//Encoder reference positions for MR4K2
nEncRefXM4K2  := ULINT_TO_UDINT(GVL_M4K2.nM4K2X_ENC_REF);
nEncRefYM4K2  := ULINT_TO_UDINT(GVL_M4K2.nM4K2Y_ENC_REF);
nEncRefrXM4K2  := ULINT_TO_UDINT(GVL_M4K2.nM4K2rX_ENC_REF);
nEncRefUSM4K2  := ULINT_TO_UDINT(GVL_M4K2.nM4K2US_ENC_REF);
nEncRefDSM4K2  := ULINT_TO_UDINT(GVL_M4K2.nM4K2DS_ENC_REF);

// M4K2 Bender Encoder Count Values For Epics
nEncCntXM4K2  := ULINT_TO_UDINT(M33.nRawEncoderULINT);
nEncCntYM4K2  := ULINT_TO_UDINT(M34.nRawEncoderULINT);
nEncCntrXM4K2  := ULINT_TO_UDINT(M35.nRawEncoderULINT);
nEncCntUSM4K2  := ULINT_TO_UDINT(M36.nRawEncoderULINT);
nEncCntDSM4K2  := ULINT_TO_UDINT(M37.nRawEncoderULINT);

// MR4K2 Bender RTDs
fM4K2US_RTD_1 := INT_TO_REAL(GVL_M4K2.nM4K2US_RTD_1);
fM4K2US_RTD_2 := INT_TO_REAL(GVL_M4K2.nM4K2US_RTD_2);
fM4K2US_RTD_3 := INT_TO_REAL(GVL_M4K2.nM4K2US_RTD_3);

fM4K2DS_RTD_1 := INT_TO_REAL(GVL_M4K2.nM4K2DS_RTD_1);


// RTD not connected if T=0
bM4K2US_RTD_1_Err := fM4K2US_RTD_1 = 0;
bM4K2US_RTD_2_Err := fM4K2US_RTD_2 = 0;
bM4K2US_RTD_3_Err := fM4K2US_RTD_3 = 0;
bM4K2DS_RTD_1_Err := fM4K2DS_RTD_1 = 0;

// M4K2 Bender RTD interlocks
M36.bHardwareEnable R= fM4K2US_RTD_1 > 9000 OR bM4K2US_RTD_1_Err;
M37.bHardwareEnable R= fM4K2DS_RTD_1 > 9000 OR bM4K2DS_RTD_1_Err;

fbM4K2_Chin_Right_RTD(fResolution:=0.01);
fbM4K2_Chin_Left_RTD(fResolution:=0.01);

// Axilon Cooling Panel
fbCoolingPanel();
(*
//PMPS
ffBenderRange.i_xOK :=
    GVL_M4K2.nM4K2US_PMPS_LowerLimit < nEncCntUSM4K2 AND nEncCntUSM4K2 < GVL_M4K2.nM4K2US_PMPS_UpperLimit AND
    GVL_M4K2.nM4K2DS_PMPS_LowerLimit < nEncCntDSM4K2 AND nEncCntUSM4K2 < GVL_M4K2.nM4K2DS_PMPS_UpperLimit;
ffBenderRange(io_fbFFHWO := GVL_PMPS.fbFastFaultOutput1);
*)
fbXSetup(stPositionState:=GVL_States.stDefaultKBX, bSetDefault:=TRUE);

fbXSetup(stPositionState:=astCoatingStatesX[E_B4C_Rh_CoatingStates.B4C],
    sName:='B4C',
    sPmpsState:='MR4K2:KBV-B4C',
    nEncoderCount:=5824240,
    fDelta:=5
);
fbXSetup(stPositionState:=astCoatingStatesX[E_B4C_Rh_CoatingStates.Rh],
    sName:='Rh',
    sPmpsState:='MR4K2:KBV-RHODIUM',
    nEncoderCount:=3524222,
    fDelta:=1.5
);
fbCoatingStates(
    stMotionStage:=Main.M33,
    astPositionState:=astCoatingStatesX,
    eEnumSet:=eStateSet,
    eEnumGet:=eStateGet,
    fbFFHWO:=GVL_PMPS.fbFastFaultOutput2,
    fbArbiter:=GVL_PMPS.fbArbiter2,
    bEnableMotion:=TRUE,
    bEnableBeamParams:=TRUE,
    sDeviceName:='MR4K2:KBV',
    sTransitionKey:='MR4K2:KBV-TRANSITION',
);

END_PROGRAM

// ---- POUs/Serial Comm/P_Serial_Com.TcPOU
PROGRAM P_Serial_Com
VAR
    fbSerialLineControl_EL6001_M1K2: SerialLineControl;
END_VAR

//These are the global IOs...don't forget to copy your data into them

(* EL6001 Serial port 0 com function *)
fbSerialLineControl_EL6001_M1K2(Mode:= SERIALLINEMODE_EL6_22B (*SERIALLINEMODE_KL6_22B_STANDARD*),
                                pComIn:= ADR(Serial_stComIn_M1K2),
                                   pComOut:=ADR(Serial_stComOut_M1K2),
                                SizeComIn:= SIZEOF(Serial_stComIn_M1K2),
                                TxBuffer:= Serial_TXBuffer_M1K2,
                                RxBuffer:= Serial_RXBuffer_M1K2,
                                Error=> ,
                                ErrorID=> );

END_PROGRAM

// ---- POUs/PRG_Stats.TcPOU
PROGRAM PRG_Stats
VAR
    // SP1K1 Grating Mono Vibration Stats
    fGpiEncoderPosDiff: LREAL;
    afGpiPosDiffBuffer: ARRAY[1..1000] OF LREAL;
    afGpiExtraBuffer: ARRAY[1..1000] OF LREAL;
    fbGpiPosDiffCollect: FB_DataBuffer;
    {attribute 'pytmc' := '
        pv: SP1K1:MONO:MMS:G_PI:ENCDIFF
    '}
    fbGpiPosDiffStats: FB_BasicStats;

    fGpiRangeMax: LREAL;
    rtNewGpiMove: R_TRIG;
    tonNewGpiMove: TON;


    // SP1K1 Mirror Pitch Mono Vibration Stats
    fMpiEncoderPosDiff: LREAL;
    afMpiPosDiffBuffer: ARRAY[1..1000] OF LREAL;
    afMpiExtraBuffer: ARRAY[1..1000] OF LREAL;
    fbMpiPosDiffCollect: FB_DataBuffer;
    {attribute 'pytmc' := '
        pv: SP1K1:MONO:MMS:M_PI:ENCDIFF
    '}
    fbMpiPosDiffStats: FB_BasicStats;


    // MR1K1 Pitch Vibration Stats
    fMR1K1PiEncoderPosDiff: LREAL;
    afMR1K1PiPosDiffBuffer: ARRAY[1..1000] OF LREAL;
    afMR1K1PiExtraBuffer: ARRAY[1..1000] OF LREAL;
    fbMR1K1PiPosDiffCollect: FB_DataBuffer;
    {attribute 'pytmc' := '
        pv: MR1K1:BEND:MMS:PITCH:ENCDIFF
    '}
    fbMR1K1PiPosDiffStats: FB_BasicStats;
END_VAR

IF rtNewGpiMove.Q THEN
    // Reset before a move
    fGpiRangeMax := 0;
ELSIF tonNewGpiMove.Q AND ABS(M7.fPosition - M7.stAxisStatus.fActPosition) > 5 THEN
    // Update only during moves, not at the start or end
    fGpiRangeMax := MAX(fGpiRangeMax, fbGpiPosDiffStats.fRange);
END_IF

fGpiEncoderPosDiff := ((UDINT_TO_LREAL(M7.nEncoderCount) / 150.0) - (M7.Axis.NcToPlc.SetPos - M7.stAxisParameters.fEncOffset)) * 1000;
fbGpiPosDiffCollect(
    bExecute:=TRUE,
    pInputAdr:=ADR(fGpiEncoderPosDiff),
    iInputSize:=SIZEOF(fGpiEncoderPosDiff),
    iElemCount:=1000,
    pPartialAdr:=ADR(afGpiPosDiffBuffer),
    pOutputAdr:=ADR(afGpiExtraBuffer),
);
fbGpiPosDiffStats(
    aSignal:=afGpiPosDiffBuffer,
    bAlwaysCalc:=TRUE,
);
rtNewGpiMove(CLK:=M7.bExecute);
tonNewGpiMove(
    IN:=M7.bExecute,
    PT:=T#15s,
);

fMpiEncoderPosDiff := ((UDINT_TO_LREAL(M6.nEncoderCount) * 0.004505) - (M6.Axis.NcToPlc.SetPos - M6.stAxisParameters.fEncOffset)) * 1000;
fbMpiPosDiffCollect(
    bExecute:=TRUE,
    pInputAdr:=ADR(fMpiEncoderPosDiff),
    iInputSize:=SIZEOF(fMpiEncoderPosDiff),
    iElemCount:=1000,
    pPartialAdr:=ADR(afMpiPosDiffBuffer),
    pOutputAdr:=ADR(afMpiExtraBuffer),
);
fbMpiPosDiffStats(
    aSignal:=afMpiPosDiffBuffer,
    bAlwaysCalc:=TRUE,
);

fMR1K1PiEncoderPosDiff := ((UDINT_TO_LREAL(M16.nEncoderCount) * 0.00244) - (M16.Axis.NcToPlc.SetPos - M16.stAxisParameters.fEncOffset)) * 1000;
fbMR1K1PiPosDiffCollect(
    bExecute:=TRUE,
    pInputAdr:=ADR(fMR1K1PiEncoderPosDiff),
    iInputSize:=SIZEOF(fMR1K1PiEncoderPosDiff),
    iElemCount:=1000,
    pPartialAdr:=ADR(afMR1K1PiPosDiffBuffer),
    pOutputAdr:=ADR(afMR1K1PiExtraBuffer),
);
fbMR1K1PiPosDiffStats(
    aSignal:=afMR1K1PiPosDiffBuffer,
    bAlwaysCalc:=TRUE,
);

END_PROGRAM

// ---- Implicit Checks/CheckBounds.TcPOU
// Implicitly generated code : DO NOT EDIT
FUNCTION CheckBounds : DINT
VAR_INPUT
    index, lower, upper: DINT;
END_VAR

// Implicitly generated code : Only an Implementation suggestion
{noflow}
IF  index < lower THEN
    CheckBounds := lower;
ELSIF  index > upper THEN
    CheckBounds := upper;
ELSE
    CheckBounds := index;
END_IF
{flow}

END_FUNCTION

// ---- Implicit Checks/CheckDivDInt.TcPOU
// Implicitly generated code : DO NOT EDIT
FUNCTION CheckDivDInt : DINT
VAR_INPUT
    divisor:DINT;
END_VAR

// Implicitly generated code : Only an Implementation suggestion
{noflow}
IF divisor = 0 THEN
    CheckDivDInt:=1;
ELSE
    CheckDivDInt:=divisor;
END_IF;
{flow}

END_FUNCTION

// ---- Implicit Checks/CheckDivLInt.TcPOU
// Implicitly generated code : DO NOT EDIT
FUNCTION CheckDivLInt : LINT
VAR_INPUT
    divisor:LINT;
END_VAR

// Implicitly generated code : Only an Implementation suggestion
{noflow}
IF divisor = 0 THEN
    CheckDivLInt:=1;
ELSE
    CheckDivLInt:=divisor;
END_IF;
{flow}

END_FUNCTION

// ---- Implicit Checks/CheckDivLReal.TcPOU
// Implicitly generated code : DO NOT EDIT
FUNCTION CheckDivLReal : LREAL
VAR_INPUT
    divisor:LREAL;
END_VAR

// Implicitly generated code : Only an Implementation suggestion
{noflow}
IF divisor = 0 THEN
    CheckDivLReal:=1;
ELSE
    CheckDivLReal:=divisor;
END_IF;
{flow}

END_FUNCTION

// ---- Implicit Checks/CheckDivReal.TcPOU
// Implicitly generated code : DO NOT EDIT
FUNCTION CheckDivReal : REAL
VAR_INPUT
    divisor:REAL;
END_VAR

// Implicitly generated code : Only an Implementation suggestion
{noflow}
IF divisor = 0 THEN
    CheckDivReal:=1;
ELSE
    CheckDivReal:=divisor;
END_IF;
{flow}

END_FUNCTION

// ---- Implicit Checks/CheckLRangeSigned.TcPOU
// Implicitly generated code : DO NOT EDIT
FUNCTION CheckLRangeSigned : LINT
VAR_INPUT
    value, lower, upper: LINT;
END_VAR

// Implicitly generated code : Only an Implementation suggestion
{noflow}
IF (value < lower) THEN
    CheckLRangeSigned := lower;
ELSIF(value > upper) THEN
    CheckLRangeSigned := upper;
ELSE
    CheckLRangeSigned := value;
END_IF

{flow}

END_FUNCTION

// ---- Implicit Checks/CheckLRangeUnsigned.TcPOU
// Implicitly generated code : DO NOT EDIT
FUNCTION CheckLRangeUnsigned : ULINT
VAR_INPUT
    value, lower, upper: ULINT;
END_VAR

// Implicitly generated code : Only an Implementation suggestion
{noflow}
IF (value < lower) THEN
    CheckLRangeUnsigned := lower;
ELSIF(value > upper) THEN
    CheckLRangeUnsigned := upper;
ELSE
    CheckLRangeUnsigned := value;
END_IF
{flow}

END_FUNCTION

// ---- Implicit Checks/CheckPointer.TcPOU
// Implicitly generated code : DO NOT EDIT
FUNCTION CheckPointer : POINTER TO BYTE
VAR_INPUT
    ptToTest : POINTER TO BYTE; // Destination address of the pointer
    iSize : DINT;		        // Size of the type the pointer points to. (e.g: 20 for POINTER TO ARRAY [0..9] OF INT)
    iGran : DINT;		        // Granularity of the pointer access. This is the size of the biggest non-structured data type in the type the pointer points to. (e.g: 2 for POINTER TO ARRAY [0..9] OF INT)
    bWrite: BOOL;		        // Indicates read or write Access. TRUE = write access.
END_VAR

// No standard way of implementation. Fill your own code here
CheckPointer := ptToTest;
{flow}

END_FUNCTION

// ---- Implicit Checks/CheckRangeSigned.TcPOU
// Implicitly generated code : DO NOT EDIT
FUNCTION CheckRangeSigned : DINT
VAR_INPUT
    value, lower, upper: DINT;
END_VAR

// Implicitly generated code : Only an Implementation suggestion
{noflow}
IF (value < lower) THEN
    CheckRangeSigned := lower;
ELSIF(value > upper) THEN
    CheckRangeSigned := upper;
ELSE
    CheckRangeSigned := value;
END_IF
{flow}

END_FUNCTION

// ---- Implicit Checks/CheckRangeUnsigned.TcPOU
// Implicitly generated code : DO NOT EDIT
FUNCTION CheckRangeUnsigned : UDINT
VAR_INPUT
    value, lower, upper: UDINT;
END_VAR

// Implicitly generated code : Only an Implementation suggestion
{noflow}
IF (value < lower) THEN
    CheckRangeUnsigned := lower;
ELSIF(value > upper) THEN
    CheckRangeUnsigned := upper;
ELSE
    CheckRangeUnsigned := value;
END_IF
{flow}

END_FUNCTION

// ---- POUs/PRG_SPO_PMPS.TcPOU
PROGRAM PRG_SPO_PMPS
VAR
    // PMPS
    ffMR1K1Height : FB_FastFault := (
        i_xAutoReset := TRUE,
        i_DevName := 'MR1K1 Height',
        i_Desc := 'MR1K1 Height is out of Single Point Operation safe range',
        i_TypeCode := 16#F501);
    ffMR1K1Pitch : FB_FastFault := (
        i_xAutoReset := TRUE,
        i_DevName := 'MR1K1 Pitch',
        i_Desc := 'MR1K1 Pitch is out of Single Point Operation safe range',
        i_TypeCode := 16#F502);

    ffSP1K1MPitch : FB_FastFault := (
        i_xAutoReset := TRUE,
        i_DevName := 'SP1K1 Mirror Pitch',
        i_Desc := 'SP1K1 Mirror Pitch is out of Single Point Operation safe range',
        i_TypeCode := 16#F503);
    ffSP1K1GPitch : FB_FastFault := (
        i_xAutoReset := TRUE,
        i_DevName := 'SP1K1 Grating Pitch',
        i_Desc := 'SP1K1 Grating Pitch is out of Single Point Operation safe range',
        i_TypeCode := 16#F504);
    ffSP1K1GHorisontal : FB_FastFault := (
        i_xAutoReset := TRUE,
        i_DevName := 'SP1K1 Grating horizontal',
        i_Desc := 'SP1K1 horizontal Pitch is out of Single Point Operation safe range',
        i_TypeCode := 16#F505);

    ffZos : FB_FastFault := (
        i_xAutoReset := TRUE,
        i_DevName := 'T1K1 ZOS',
        i_Desc := 'ST1K1 ZOS is out of Single Point Operation safe range',
        i_TypeCode := 16#F506);
END_VAR
VAR CONSTANT
    nUpperMR1K1Height : UDINT := 32961458; //POS 32911458+ Delta 50000;
    nLowerMR1K1Height : UDINT := 32861458; //POS 32911458- Delta 50000;

    nUpperMR1K1Pitch : UDINT := 10114377;// 10093885 + 20491;
    nLowerMR1K1Pitch : UDINT := 10073393; //10093885 - 20491;

    nUpperSP1K1MPitch : UDINT := 31769145;// 31758046 + 11098;
    nLowerSP1K1MPitch : UDINT := 31746947;//31758046 - 11098;

    nUpperSP1K1MPitch_400 : UDINT := 31285238;
    nLowerSP1K1MPitch_400 : UDINT := 31263041;

    nUpperSP1K1MPitch_1000 : UDINT := 31809544;
    nLowerSP1K1MPitch_1000 : UDINT := 31787347;

    nUpperSP1K1GPitch_700 : UDINT := 23624881;
    nUpperSP1K1GPitch_400 : UDINT := 23204883;
    nUpperSP1K1GPitch_1000 : UDINT := 23564882;

    nUpperSP1K1GH: UDINT := 40000000;
    nLowerSP1K1GH: UDINT := 24000000;

    nZOSLower : UDINT := 22926596; // value still needs to be verified


END_VAR


IF (GVL_PMPS.rPhotonEnergy < 715) AND (GVL_PMPS.rPhotonEnergy >685) THEN
    ffSP1K1MPitch.i_xOK := PRG_MR1K1_BEND_BENDER.ffBenderRange.i_xOK OR ((M6.nEncoderCount > nLowerSP1K1MPitch) AND (M6.nEncoderCount < nUpperSP1K1MPitch));
    ffSP1K1GPitch.i_xOK := PRG_MR1K1_BEND_BENDER.ffBenderRange.i_xOK OR ((M7.nEncoderCount < nUpperSP1K1GPitch_700));
ELSIF (GVL_PMPS.rPhotonEnergy < 410) AND (GVL_PMPS.rPhotonEnergy >390) THEN
    ffSP1K1MPitch.i_xOK := PRG_MR1K1_BEND_BENDER.ffBenderRange.i_xOK OR ((M6.nEncoderCount > nLowerSP1K1MPitch_400) AND (M6.nEncoderCount < nUpperSP1K1MPitch_400));
    ffSP1K1GPitch.i_xOK := PRG_MR1K1_BEND_BENDER.ffBenderRange.i_xOK OR ((M7.nEncoderCount < nUpperSP1K1GPitch_400));
ELSIF (GVL_PMPS.rPhotonEnergy < 1020) AND (GVL_PMPS.rPhotonEnergy >980) THEN
    ffSP1K1MPitch.i_xOK := PRG_MR1K1_BEND_BENDER.ffBenderRange.i_xOK OR ((M6.nEncoderCount > nLowerSP1K1MPitch_1000) AND (M6.nEncoderCount < nUpperSP1K1MPitch_1000));
    ffSP1K1GPitch.i_xOK := PRG_MR1K1_BEND_BENDER.ffBenderRange.i_xOK OR ((M7.nEncoderCount < nUpperSP1K1GPitch_1000));
ELSE
    ffSP1K1MPitch.i_xOK := PRG_MR1K1_BEND_BENDER.ffBenderRange.i_xOK;
    ffSP1K1GPitch.i_xOK := PRG_MR1K1_BEND_BENDER.ffBenderRange.i_xOK;

END_IF


//MR1K1 height
ffMR1K1Height.i_xOK := PRG_MR1K1_BEND_BENDER.ffBenderRange.i_xOK OR ((M12.nEncoderCount > nLowerMR1K1Height ) AND (M12.nEncoderCount < nUpperMR1K1Height ));
ffMR1K1Height(io_fbFFHWO := GVL_PMPS.fbFastFaultOutput1);
//MR1K1 pitch
ffMR1K1Pitch.i_xOK := PRG_MR1K1_BEND_BENDER.ffBenderRange.i_xOK OR ( (M16.nEncoderCount > nLowerMR1K1Pitch) AND ( M16.nEncoderCount < nUpperMR1K1Pitch));
ffMR1K1Pitch(io_fbFFHWO := GVL_PMPS.fbFastFaultOutput1);
//SP1K1 mirror pitch
ffSP1K1MPitch(io_fbFFHWO := GVL_PMPS.fbFastFaultOutput1);
//SP1K1 grating pitch
ffSP1K1GPitch(io_fbFFHWO := GVL_PMPS.fbFastFaultOutput1);
//SP1K1 Grating horizontal
ffSP1K1GHorisontal.i_xOK := PRG_MR1K1_BEND_BENDER.ffBenderRange.i_xOK OR ((M9.nEncoderCount > nLowerSP1K1GH) AND (M9.nEncoderCount < nUpperSP1K1GH));
ffSP1K1GHorisontal(io_fbFFHWO := GVL_PMPS.fbFastFaultOutput1);
//ST1K1 ZOS
ffZos.i_xOK := PRG_MR1K1_BEND_BENDER.ffBenderRange.i_xOK OR (M24.nEncoderCount <= nZOSLower); //encoder counts decreases as value in mm increases
ffZos(io_fbFFHWO := GVL_PMPS.fbFastFaultOutput1);

END_PROGRAM
